PROGRAM prgRWEffIO
VAR
	fbRW1		: FB_ReadWrite_V2;
END_VAR

fbRW1(eUploadType := eSelectDataUploadType.e_Change_Intervall5min, bBusy=> , bError=> , udiErrorCodeOut=> , eErrorReadWrite_Out=> );

END_PROGRAM

(* stored: Version 1.1.0.1, ProductVersion 3.1.4024.12
   POU prgRWEffIO: Id {785bf272-28fb-4849-abf1-556c1eb322b8}, SpecialFunc None *)
